FUNCTION_BLOCK shift (* Composite Function Block Type *)
  (* Standard: 61499-2 *)
  (* Version 0.2, 2003-12-05, JHC, Rockwell Automation, Renamed from NEWCOMPFB. *)
  (* Version 0.1, 2002-01-08, JHC, Rockwell Automation, Added DLY FB as example. *)
  (* Version 0.0, 2000-05-27, JHC, Rockwell Automation *)
  (* Compiler header: package fb.rt.pnp; import fb.rt.vmath.*; *)
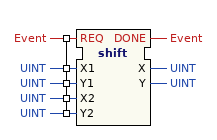
  EVENT_INPUT
    REQ WITH X1, Y1, X2, Y2; (* Normal Execution Request *)
  END_EVENT
  EVENT_OUTPUT
    DONE;
  END_EVENT
  VAR_INPUT
    X1 : UINT;
    Y1 : UINT;
    X2 : UINT;
    Y2 : UINT;
  END_VAR
  VAR_OUTPUT
    X : UINT;
    Y : UINT;
  END_VAR
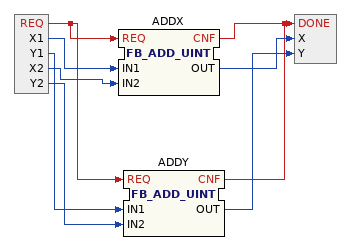
  FBS
    ADDX : FB_ADD_UINT;
    ADDY : FB_ADD_UINT;
  END_FBS
  EVENT_CONNECTIONS
    ADDX.CNF TO DONE;
    REQ TO ADDX.REQ;
    REQ TO ADDY.REQ;
    ADDY.CNF TO DONE;
  END_CONNECTIONS
  DATA_CONNECTIONS
    X1 TO ADDX.IN1;
    X2 TO ADDX.IN2;
    ADDX.OUT TO X;
    Y1 TO ADDY.IN1;
    Y2 TO ADDY.IN2;
    ADDY.OUT TO Y;
  END_CONNECTIONS
END_FUNCTION_BLOCK
